{attribute 'GeneratedUsingTerminal: ER7342-0002-0020'}
{attribute addProperty BoxType "ER7342-0002-0020"}
{attribute addProperty Id "ControlAT %Q*Control_C948E0F23"}
{attribute addProperty CRC "1519079446"}
{attribute addProperty Size "3"}
TYPE DCM_Control_Channel_5A8B5016 EXTENDS OutputBase_10CEE7DE :
STRUCT
	{attribute addProperty Name "Control"}
	Control AT %Q* : Control_C948E0F2;
END_STRUCT
END_TYPE

(* stored: Version 1.2.0.0, ProductVersion 3.1.4024.9
   DUT DCM_Control_Channel_5A8B5016: Id {d31873ce-eb02-4dc0-9003-deef8bb49fa0} *)
